PROGRAM PRG_4_LOG
VAR
    fbLogHandler: FB_LogHandler;
END_VAR

fbLogHandler();

END_PROGRAM

(* stored: Version 1.1.0.1, ProductVersion 3.1.4022.18
   POU PRG_4_LOG: Id {f3d0f566-4bb2-4598-97b7-7f257847c644}, SpecialFunc None *)
